// LS Electric XG5000 project: PLC_최종프로젝트 프로그램
// PLC LSPLC
// module base 0 slot 0: 입출력 모듈:XBC-DR32H (DC 24V 입력, 릴레이 출력 32점)

PROGRAM 01_Conveyor_Belt (task: 스캔 프로그램)

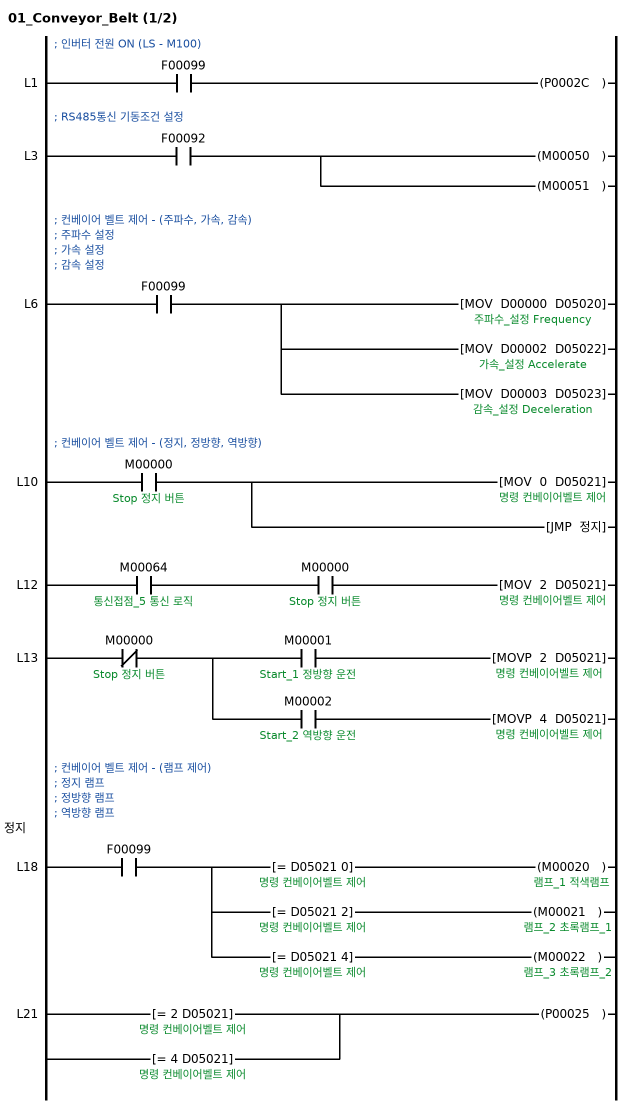
// 인버터 전원 ON (LS - M100)
; L1
LOAD      F00099
OUT       P0002C
// RS485통신 기동조건 설정
; L3
LOAD      F00092
OUT       M00050
OUT       M00051
// 컨베이어 벨트 제어 - (주파수, 가속, 감속)
; L6
LOAD      F00099
MOV       D00000 D05020	// 주파수_설정 Frequency
MOV       D00002 D05022	// 가속_설정 Accelerate
MOV       D00003 D05023	// 감속_설정 Deceleration
// output comment: 주파수 설정
// output comment: 가속 설정
// output comment: 감속 설정
// 컨베이어 벨트 제어 - (정지, 정방향, 역방향)
; L10
LOAD      M00000	// Stop 정지 버튼
MOV       0 D05021	// 명령 컨베이어벨트 제어
JMP       정지
; L12
LOAD      M00064	// 통신접점_5 통신 로직
AND       M00000	// Stop 정지 버튼
MOV       2 D05021	// 명령 컨베이어벨트 제어
; L13
LOAD NOT  M00000	// Stop 정지 버튼
MPUSH
AND       M00001	// Start_1 정방향 운전
MOVP      2 D05021	// 명령 컨베이어벨트 제어
MPOP
AND       M00002	// Start_2 역방향 운전
MOVP      4 D05021	// 명령 컨베이어벨트 제어
정지:
// 컨베이어 벨트 제어 - (램프 제어)
; L18
LOAD      F00099
MPUSH
AND=      D05021 0	// 명령 컨베이어벨트 제어
OUT       M00020	// 램프_1 적색램프
MLOAD
AND=      D05021 2	// 명령 컨베이어벨트 제어
OUT       M00021	// 램프_2 초록램프_1
MPOP
AND=      D05021 4	// 명령 컨베이어벨트 제어
OUT       M00022	// 램프_3 초록램프_2
// output comment: 정지 램프
// output comment: 정방향 램프
// output comment: 역방향 램프
; L21
LOAD=     2 D05021	// 명령 컨베이어벨트 제어
OR=       4 D05021	// 명령 컨베이어벨트 제어
OUT       P00025

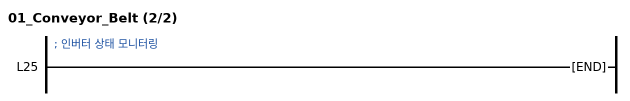
// 인버터 상태 모니터링
; L25
END

PROGRAM 02_Sensor (task: 스캔 프로그램)

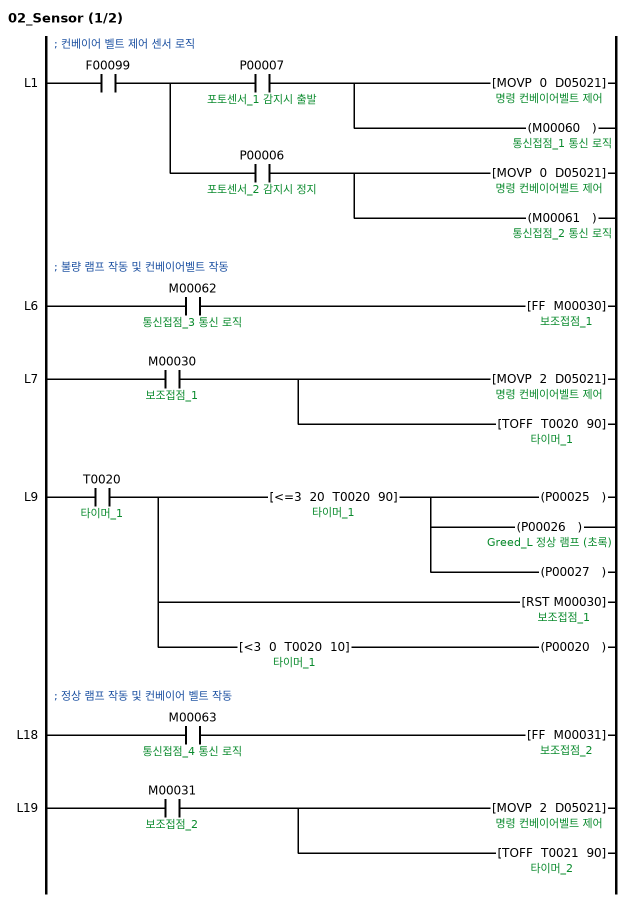
// 컨베이어 벨트 제어 센서 로직
; L1
LOAD      F00099
MPUSH
AND       P00007	// 포토센서_1 감지시 출발
MOVP      0 D05021	// 명령 컨베이어벨트 제어
OUT       M00060	// 통신접점_1 통신 로직
MPOP
AND       P00006	// 포토센서_2 감지시 정지
MOVP      0 D05021	// 명령 컨베이어벨트 제어
OUT       M00061	// 통신접점_2 통신 로직
// 불량 램프 작동 및 컨베이어벨트 작동
; L6
LOAD      M00062	// 통신접점_3 통신 로직
FF        M00030	// 보조접점_1
; L7
LOAD      M00030	// 보조접점_1
MOVP      2 D05021	// 명령 컨베이어벨트 제어
TOFF      T0020 90	// 타이머_1
; L9
LOAD      T0020	// 타이머_1
MPUSH
AND<=3    20 T0020 90	// 타이머_1
OUT       P00025
OUT       P00026	// Greed_L 정상 램프 (초록)
OUT       P00027
MPOP
RST       M00030	// 보조접점_1
AND<3     0 T0020 10	// 타이머_1
OUT       P00020
// 정상 램프 작동 및 컨베이어 벨트 작동
; L18
LOAD      M00063	// 통신접점_4 통신 로직
FF        M00031	// 보조접점_2
; L19
LOAD      M00031	// 보조접점_2
MOVP      2 D05021	// 명령 컨베이어벨트 제어
TOFF      T0021 90	// 타이머_2

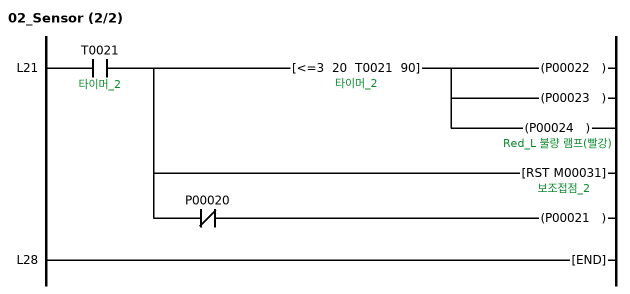
; L21
LOAD      T0021	// 타이머_2
MPUSH
AND<=3    20 T0021 90	// 타이머_2
OUT       P00022
OUT       P00023
OUT       P00024	// Red_L 불량 램프(빨강)
MPOP
RST       M00031	// 보조접점_2
AND NOT   P00020
OUT       P00021
; L28
END

PROGRAM 03_Modbus_통신 (task: 스캔 프로그램)

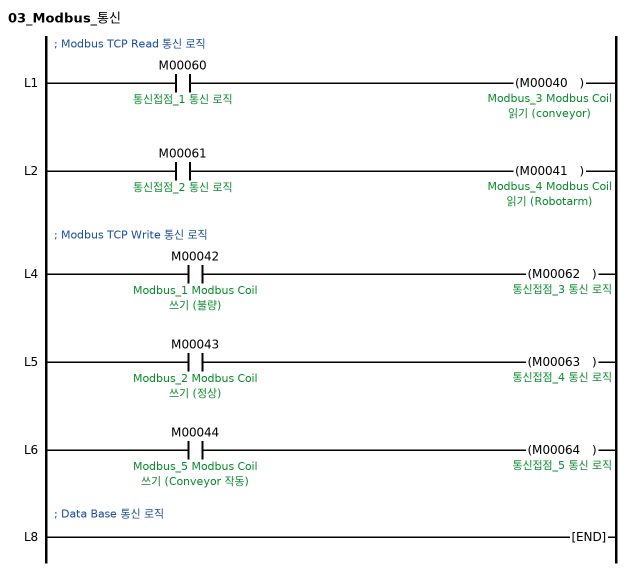
// Modbus TCP Read 통신 로직
; L1
LOAD      M00060	// 통신접점_1 통신 로직
OUT       M00040	// Modbus_3 Modbus Coil 읽기 (conveyor)
; L2
LOAD      M00061	// 통신접점_2 통신 로직
OUT       M00041	// Modbus_4 Modbus Coil 읽기 (Robotarm)
// Modbus TCP Write 통신 로직
; L4
LOAD      M00042	// Modbus_1 Modbus Coil 쓰기 (불량)
OUT       M00062	// 통신접점_3 통신 로직
; L5
LOAD      M00043	// Modbus_2 Modbus Coil 쓰기 (정상)
OUT       M00063	// 통신접점_4 통신 로직
; L6
LOAD      M00044	// Modbus_5 Modbus Coil 쓰기 (Conveyor 작동)
OUT       M00064	// 통신접점_5 통신 로직
// Data Base 통신 로직
; L8
END

VARIABLES AND COMMENTS (devices not used above)
M00004	BIT	Select_버튼 // 수동/자동
M00015	BIT	Start_Bt // 자동 시작 버튼
M00016	BIT	Start_Stop // 시작 / 정지
M00017	BIT	Stop_Bt // 자동 정지 버튼
D04970	WORD	가속_입력 // Accelerate
D04980	WORD	감속_입력 // Deceleration
M00032	BIT	보조접점_3
M00033	BIT	보조접점_4
M00034	BIT	보조접점_5
M00035	BIT	보조접점_6
M00005	BIT	수동_자동 // 수동 및 자동 제어
M00006	BIT	자동 // 자동 제어
D04960	WORD	주파수_입력 // Frequency
T0001	BIT/WORD	타미어_4
T0002	BIT/WORD	타미어_5
T0003	BIT/WORD	타미어_6
T0000	BIT/WORD	타이머_3